// TIA Portal V17 export
// export: Created 2022-05-07T16:38:48.6865755Z, ExportSetting WithDefaults, DisplayName Totally Integrated Automation Portal, DisplayVersion V17 Update 3, DisplayName TIA Portal Openness, DisplayVersion V17 Update 3, DisplayName TIA Portal Version Control Interface, DisplayVersion V17, DisplayName TIA Portal Test Suite Advanced, DisplayVersion V17 Update 1, DisplayName SINAMICS Startdrive Advanced, DisplayVersion V17 Update2, DisplayName SINAMICS Startdrive G130, G150, S120, S150, SINAMICS MV, S210, DisplayVersion V17 Update2, DisplayName SINAMICS Startdrive G110M, G120, G120C, G120D, G120P, G115D, DisplayVersion V17 Update2, DisplayName STEP 7 Professional, DisplayVersion V17 Update 3, DisplayName STEP 7 Safety, DisplayVersion V17, DisplayName WinCC UA Professional, DisplayVersion V17 Update 3
DATA_BLOCK "FB_PosizAsseStandard_DB"   // DB5
VERSION : 0.1
// stored: AutoNumber true, DBAccessibleFromOPCUA true, InstanceOfName FB_PosizAsseStandard, InstanceOfType FB
"FB_PosizAsseStandard"
   // VAR_INPUT
   //    Exe_MC_Reset : Bool;
   //    En_MC_Power : Bool;
   //    Exe_MC_Home : Bool;
   //    Exe_Jog_Fwd : Bool;
   //    Exe_Jog_Rev : Bool;
   //    Exe_MC_Velocity : Bool;
   //    Exe_MC_Relative : Bool;
   //    Exe_MC_Abs : Bool;
   //    Exe_MC_Halt : Bool;
   //    Ctl_MC_Stop : Bool;
   //    Sp_lr_MC_HomingOffset : LReal;
   //    Sp_lr_MC_Velocity : LReal;
   //    Sp_lr_MC_RelativeDistance : LReal;
   //    Sp_lr_MC_AbsPosition : LReal;
   // END_VAR
   // VAR_OUTPUT
   //    Output_MC_At_Standstill : Bool;
   //    Output_MC_AxisEnabled : Bool;
   //    Output_MC_MoveAbs_Done : Bool;
   //    Output_MC_MoveAbs_Busy : Bool;
   //    Output_MC_Error : Bool;
   //    Output_MC_AxisHomed : Bool;
   //    Output_ActVelocity : Real;
   //    Output_ActPos : Real;
   // END_VAR
   // VAR_IN_OUT
   //    AxisTO : TO_PositioningAxis;
   // END_VAR
   // VAR
   //    AxisReady_PosAxis { S7_SetPoint := 'True'} : Bool;
   //    MC_Power_Instance_1 { S7_SetPoint := 'True'} : MC_Power;
   //    MC_Home_Instance_1 { S7_SetPoint := 'True'} : MC_Home;
   //    MC_MoveJog_Instance_1 { S7_SetPoint := 'True'} : MC_MoveJog;
   //    MC_MoveVelocity_Instance_1 { S7_SetPoint := 'True'} : MC_MoveVelocity;
   //    MC_MoveRelative_Instance_1 { S7_SetPoint := 'True'} : MC_MoveRelative;
   //    MC_MoveAbsolute_Instance_1 { S7_SetPoint := 'True'} : MC_MoveAbsolute;
   //    MC_Halt_Instance_1 { S7_SetPoint := 'True'} : MC_Halt;
   //    MC_Reset_Instance_1 { S7_SetPoint := 'True'} : MC_Reset;
   // END_VAR
BEGIN
END_DATA_BLOCK
